(* 캠트리거 파이프라인 — 파이버 센서 감지부터 카메라 트리거까지 (연속 리얼타임).
   전단(리딩엣지=상승엣지)에서 엔코더 기준점을 큐에 push. 유효조건: rising 직전에
   OFF 가 PRE_OFF_STABLE 연속 유지(무장) — 부품 중간/꼬리의 반사 깜빡임 rising 은
   직전 OFF 가 짧아 부품 길이와 무관하게 차단됨 →
   head 기준점 + Trigger_Length 도달 시 1회 트리거 + pop. 오토모드 전용.
   ⚠ 기준점이 후단→전단으로 변경됨: Trigger_Length(Cam_Trigger_Length) 는
     리딩엣지 기준 거리로 재튜닝 필요(기존값 + 부품 길이 만큼 커져야 같은 지점 촬영).
   (수동/마스터링 캠트리거는 Mastering.TcPOU 에서 별도 구동)

   pop 안전장치:
     - 위치 불연속(엔코더 리셋·대형 역행 점프) 시 큐 flush(stale head 방지)
     - Reset(시스템초기화/사이클말) 시 큐 비움 *)
FUNCTION_BLOCK FB_CamTrigger
VAR_INPUT
    Auto_Mode      : BOOL;     // 오토모드(미오토 시 큐 flush + 트리거 정지)
    Fiber_Sensor   : BOOL;     // 파이버 센서 입력
    Real_Position  : LREAL;    // 엔코더 실제 위치
    Conveyor_CCW   : BOOL;     // 컨베이어 역방향(큐 flush)
    Trigger_Length : LREAL;    // 기준점 + 이 거리 도달 시 트리거(GVL_Vision.Cam_Trigger_Length)
    Reset          : BOOL;     // 시스템초기화/사이클말 큐 비움(레벨, 상승엣지에 1회 clear)
END_VAR
VAR_OUTPUT
    Trigger        : BOOL;     // 0.1s 정형된 캠트리거 펄스(오토 발동분)
    Trig_Position  : LREAL;    // 트리거 순간 엔코더 위치 래치(Target X 보정 기준)
END_VAR
VAR
    Rise_Trig          : R_TRIG;            // 센서 상승엣지(전단=리딩엣지 감지)
    Off_Stable         : TON;               // rising 유효조건: 직전에 OFF 가 PRE_OFF_STABLE 연속 유지됐어야 함.
                                            // 부품 중간 깜빡임 rising 은 직전 OFF 가 수십 ms 뿐 → 부품 어디서 깜빡여도 차단.
    Armed              : BOOL;              // OFF 안정 확인됨 → 다음 rising 을 진짜 리딩엣지로 인정
    PRE_OFF_STABLE     : TIME := T#150MS;   // 제약: < 부품간 OFF 시간(30mm/130mm/s=0.23s, 35% 여유)
                                            //       > 깜빡임 최대 OFF 폭(통상 수십 ms)
    Trig_Pulse         : TP;                // 0.1s 펄스 정형
    Reset_Trig         : R_TRIG;            // Reset 상승엣지
    bDistReached       : BOOL;              // 이번 스캔 head 가 촬영거리 도달
    Last_Real_Position : LREAL;             // 직전 스캔 엔코더 위치(위치 불연속 감지용)
    Queue              : FB_LRealRingQueue; // 캠트리거 기준점 큐(용량5)
    RESET_JUMP_MIN     : LREAL := 100;      // 역방향 점프 임계(>1스캔 최대 이송) — 엔코더 스케일 맞춰 튜닝
END_VAR

Rise_Trig(CLK := Fiber_Sensor);
Reset_Trig(CLK := Reset);

// ===== 리딩엣지 판정: '직전에 OFF 가 PRE_OFF_STABLE 연속 유지' 된 rising 만 새 부품 =====
// 부품이 센서를 가리는 동안(ON) Off_Stable 은 리셋 상태 → 부품 중간/꼬리 깜빡임 rising 은
// 직전 OFF 가 짧아 무장(Armed)이 안 되므로 부품 길이와 무관하게 차단된다.
Off_Stable(IN := NOT Fiber_Sensor, PT := PRE_OFF_STABLE);
IF Off_Stable.Q THEN
    Armed := TRUE;
END_IF
IF Auto_Mode AND Rise_Trig.Q AND Armed THEN
    Queue.Push(Real_Position);   // 리딩엣지 위치 즉시 push — 지연 0 (만재 시 유실: 용량5, 정상 흐름에선 불발생)
    Armed := FALSE;
END_IF

// ===== head 기준점 + Trigger_Length 도달 시 1회 발동 + pop =====
bDistReached := FALSE;
IF Auto_Mode
   AND Trigger_Length > 0       // 길이 오설정(0/음수) 시 과트리거 방지(pop 보호)
   AND Queue.Count > 0
   AND NOT Trig_Pulse.Q         // ★ 직전 트리거 펄스(0.1s) 진행 중엔 발동 보류.
                                //   안 그러면 펄스폭 안에 들어온 다음 부품이 pop 되며 Trig_Position 만 덮어쓰고
                                //   카메라는 안 찍히는 desync(=가까운 부품 트리거거리 부정확) 발생.
   AND (Queue.HeadValue + Trigger_Length <= Real_Position) THEN
    bDistReached := TRUE;
    Trig_Position := Real_Position;   // 실제 발동 순간 엔코더 래치 — 카메라 실촬영 위치와 1:1 일치
    Queue.Pop();
END_IF

// 0.1s 펄스 정형
Trig_Pulse(IN := bDistReached, PT := T#0.1S);
Trigger := Trig_Pulse.Q;

// ===== 큐 flush =====
//  (1) 오토 이탈 / 컨베이어 역방향(Conveyor_CCW)
//  (2) 위치 불연속(엔코더 리셋 Set_Pos · 대형 역행 점프): head 기준점이 영구 도달불가가 되어
//      pop 정지 → stale 큐(Cam_Trig_Position 오류) 방지. 정상 전진/pop 시 Real 은 뒤로
//      점프하지 않으므로 오검출 없음. (RESET_JUMP_MIN 은 1스캔 최대 이송보다 크게 튜닝)
IF NOT Auto_Mode
   OR Conveyor_CCW
   OR ((Last_Real_Position - Real_Position) > RESET_JUMP_MIN) THEN
    Queue.Clear();
END_IF
Last_Real_Position := Real_Position;

// ===== 시스템 초기화 / 사이클말 큐 비움 (구 Vision_ST run7 의 큐 clear) =====
IF Reset_Trig.Q THEN
    Queue.Clear();
END_IF

END_FUNCTION_BLOCK

(* stored: Version 1.1.0.1, ProductVersion 3.1.4024.16
   POU FB_CamTrigger: Id {b2c3d4e5-0001-4b01-9101-000000000101}, SpecialFunc None *)
